FUNCTION_BLOCK fb_ratio_ctrl

VAR_INPUT
END_VAR

VAR_OUTPUT
END_VAR

VAR
	a_feed_rate_dpi: fb_flow_rate 			:= (kc:=0.01, ti:=0.001/60, Ts:=g_Ts_base, hi :=100, lo:=0, yout:=xmv_0[3]);
	d_feed_rate_dpi: fb_flow_rate 			:= (kc:=1.6E-6, ti:=0.001/60, Ts:=g_Ts_base, hi :=100, lo:=0, yout:=xmv_0[1]);
	e_feed_rate_dpi: fb_flow_rate 			:= (kc:=1.8E-6, ti:=0.001/60, Ts:=g_Ts_base, hi :=100, lo:=0, yout:=xmv_0[2]);
	c_feed_rate_dpi: fb_flow_rate 			:= (kc:=0.003, ti:=0.001/60, Ts:=g_Ts_base, hi :=100, lo:=0, yout:=xmv_0[4]);
	purge_rate_dpi: fb_flow_rate 			:= (kc:=0.01, ti:=0.001/60, Ts:=g_Ts_base, hi :=100, lo:=0, yout:=xmv_0[6]);
	separator_flow_rate_dpi: fb_flow_rate	:= (kc:=4E-4, ti:=0.001/60, Ts:=g_Ts_base, hi :=100, lo:=0, yout:=xmv_0[7]);
	stripper_flow_rate_dpi: fb_flow_rate	:= (kc:=4E-4, ti:=0.001/60, Ts:=g_Ts_base, hi :=100, lo:=0, yout:=xmv_0[8]);	
END_VAR

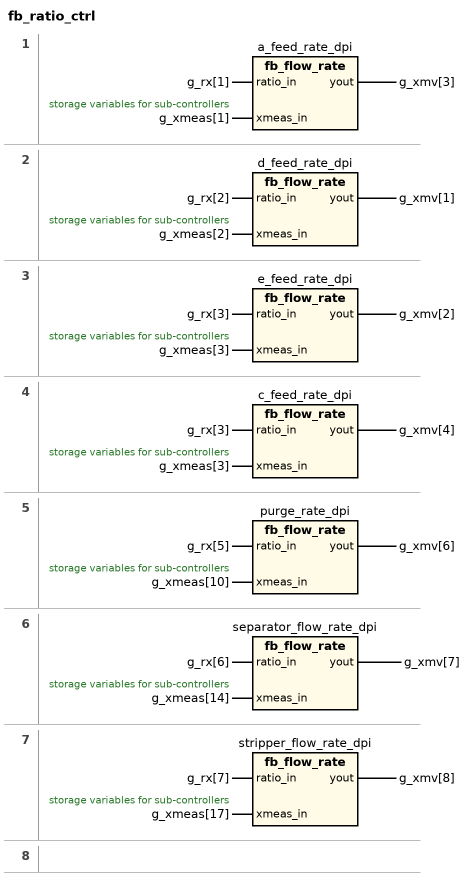
// NETWORK 1
//   g_xmeas[1]: storage variables for sub-controllers
a_feed_rate_dpi(ratio_in := g_rx[1], xmeas_in := g_xmeas[1]); // fb_flow_rate
g_xmv[3] := a_feed_rate_dpi.yout;

// NETWORK 2
//   g_xmeas[2]: storage variables for sub-controllers
d_feed_rate_dpi(ratio_in := g_rx[2], xmeas_in := g_xmeas[2]); // fb_flow_rate
g_xmv[1] := d_feed_rate_dpi.yout;

// NETWORK 3
//   g_xmeas[3]: storage variables for sub-controllers
e_feed_rate_dpi(ratio_in := g_rx[3], xmeas_in := g_xmeas[3]); // fb_flow_rate
g_xmv[2] := e_feed_rate_dpi.yout;

// NETWORK 4
//   g_xmeas[3]: storage variables for sub-controllers
c_feed_rate_dpi(ratio_in := g_rx[3], xmeas_in := g_xmeas[3]); // fb_flow_rate
g_xmv[4] := c_feed_rate_dpi.yout;

// NETWORK 5
//   g_xmeas[10]: storage variables for sub-controllers
purge_rate_dpi(ratio_in := g_rx[5], xmeas_in := g_xmeas[10]); // fb_flow_rate
g_xmv[6] := purge_rate_dpi.yout;

// NETWORK 6
//   g_xmeas[14]: storage variables for sub-controllers
separator_flow_rate_dpi(ratio_in := g_rx[6], xmeas_in := g_xmeas[14]); // fb_flow_rate
g_xmv[7] := separator_flow_rate_dpi.yout;

// NETWORK 7
//   g_xmeas[17]: storage variables for sub-controllers
stripper_flow_rate_dpi(ratio_in := g_rx[7], xmeas_in := g_xmeas[17]); // fb_flow_rate
g_xmv[8] := stripper_flow_rate_dpi.yout;

// NETWORK 8

END_FUNCTION_BLOCK

(* stored: Version 1.1.0.1, ProductVersion 3.1.0.26
   POU fb_ratio_ctrl: Id {4e39a809-28eb-4848-81f9-430c28f4d764} *)
